(*
Nazwa:			P01_PucksInserter
Opis:			Stacja podajnika opakowań
Wersja:			v0.1
Data:			2025-02-04
Autor:			DP
Urzadzenia:		
Konfiguracja:	
Info:

*)
PROGRAM P01_PucksInserter
VAR_INPUT

	//52N6.1 Pneumatyka IO
	IbPucksInserterLevelSensor					:BOOL;			// Czujnik kolejki butelki
	IbPucksInserterWheelEntrySensor				:BOOL;			// Czujnik   pierwszego slotu w karuzeli (to 
	IbPucksInserterWheelExitSensor				:BOOL;			// Czujnik
	IbPucksInserterFormGateBeforeSensor 		:BOOL;			// Czujnik przed szlabanem formatek
	IbPucksInserterFormGateAfterSensor 			:BOOL;			// Czujnik za szlabanem formatek	
 	IbPucksInserterHammerUpSensor				:BOOL;			// Czujnik położenia siłownika - góra
	IbPucksInserterHammerDownSensor				:BOOL;			// Czujnik polożenia siłowniak - dół
	IbPucksInserterTrayOnSensor					:BOOL;			// Czujnik tacka wysunieta
	//52N6.2 Pneumatyka IO	
	IbPucksInserterTrayOffSensor				:BOOL;			// Czujnik tacka schowana
	IbPucksInserterFormPositioningOnSensor		:BOOL;			// Czujnik wysuniecia siłownika pozycjonujacego formatke
	IbPucksInserterFormPositioningOffSensor		:BOOL;			// Czujnik schowania siłownika pozycjonujacego formatke
	IbPucksInserterGate1OnSensor				:BOOL;			// Czujnik otwarcia 1 szlabanu (Lewy)
	IbPucksInserterGate1OffSensor				:BOOL;			// Czujnik zamknięcia 1 szlabanu (Lewy) 
	IbPucksInserterGate2OnSensor				:BOOL;			// Czujnik otwarcia 2 szlabanu 
	IbPucksInserterGate2OffSensor				:BOOL;			// Czujnik zamknięcia 2 szlabanu (Prawy) 
	IbPucksInserterHomingSensor					:BOOL;			// Czujnik bazowania
	
	//Inne
	IbPucksInserterNotInsertedSensor			:BOOL;			// Czujnik źle włozonej butelki za stacją	
	
	IbPucksInserterPushTablesSensor				:BOOL;
END_VAR

VAR

	//BC3 
	IbPucksInserterFuseDrivesOK					AT %I*: BOOL; 			// Zabezpieczenie serwa
	IbPucksInserterTransporter1OK				AT %I*: BOOL; 			// Bezpiecznik silnikowe napędu transportera 1
	IbPucksInserterTransporter2OK				AT %I*: BOOL; 			// Bezpiecznik silnikowe napędu transportera 2	
	IbPucksInserterFuseFB1OK					AT %I*: BOOL;			// Bezpiecznik FB1 przepalony
	QbPucksInserterHammerHeightUpCmd 			AT %Q*: BOOL; 			// Wyjście sterujące podnośnikiem
	QbPucksInserterHammerHeightDownCmd 			AT %Q*: BOOL; 			// Wyjście sterujące podnośnikiem
	//GVL_IO QbPickInserterDoorsClose			AT %Q*:BOOL;			// Rozkaz zamkniecia
	QudiPucksInserterHammerHeightEncoderSetCV	AT %Q*: UDINT;			// Enkoder - Set Counter value
	QbPucksInserterHammerHeightEncoderSetC		AT %Q*: BOOL; 			// Enkoder - Set Counter 
	IudiPucksInserterHammerHeightEncoderCV 		AT %I*: UDINT;	 		// Enkoder - Counter value
	IbPucksInserterHammerHeightEncoderSetCDone	AT %I*: BOOL; 			// Enkoder - Set Counter done

	//DI5
	//GVL_IO IbPucksInserterDoorsOpen	{warning 'PI'}	AT %I*	:BOOL;	//Otwarte drzwi podajnika opakowań
	//GLV_IO etop 0
	//GLV_IO etop 1
	//GLV_IO stop
	//GLV_IO start
	//Safety reset

	//DO4
	//Lamps green
	//Lamps blue

	fbPucksInserter						  	: FB_PucksInserter;		// Bloczek do obsługi stacji podajnika butelek
	fbTurnTable								: FB_MitsubishiInverter; 	//Bloczek do obsługi falownika stołu obrotewego
	
	ePucksInserterStationState				: E_Station;
	ePucksInserterRunningState				: E_PuckInserterState;
	fbPucksInserterState					: FB_State;
	
	ePucksInserterTurnTableState			: E_Station;
	ePucksInserterTurnTableRunningState		: E_ConveyorState;
	fbBottleSorterTurnTableState			: FB_State;
	
	fbGatePucksInserter						: FB_SpringGateV2;
	
	//Wyjścia sterujące
	QbPucksInserterHammer					:BOOL;			// Wbijak
	QbPucksInserterTray						:BOOL;			// Ruchomy blat (tacka)
	QbPucksInserterGate1					:BOOL;			// Szlaban 1 (lewy)
	QbPucksInserterGate2					:BOOL;			// Szlaban 2 (prawy)
	QbPucksInserterFormGate					:BOOL;			// Szlaban formatki
	QbPucksInserterFormPositioning			:BOOL;			// Pozycjonowanie formatki

	// Stół obrotowy
	uiPucksInserterTurnTableSW					AT %I*: UINT;
	uiPucksInserterTurnTableActualVelocity		AT %I*: UDINT;
	uiPucksInserterTurnTableCW  				AT %Q*: UINT;
	udiPucksInserterTurnTableVelocity			AT %Q*: UDINT;
	
	// Transporter
	uiPucksInserterConveyorSW					AT %I*: UINT;
	uiPucksInserterConveyorActualVelocity		AT %I*: UDINT;
	uiPucksInserterConveyorCW  					AT %Q*: UINT;
	udiPucksInserterConveyorVelocity			AT %Q*: UDINT;	
	IbPucksInserterConveyorWcState				AT %I*: BOOL;
	
	// Serwo
	// GVL axis
	diPucksInserterWheelZPhaseOffset			AT %I*: DINT; // Offset serwa Z


	// Bazowanie
	tonPucksInserterEnable	: TON;
	rtEnable	: R_TRIG;
	
	//testowe
	bTest :BOOL;
	bTest2 :BOOL;	
	bTestHomingPI:BOOL;
	bPITest:BOOL;
	 
	//Stół pchający    //Vasyl 27.05
	fbPushTable_m1: FB_MitsubishiInverter;
	fbPushTable_m2: FB_MitsubishiInverter;
	fbPushTable_m3: FB_MitsubishiInverter;	
	
	QnPucksInserterPushTable_m1_VelocitySV 						AT %Q*: UDINT; 	
	InPucksInserterPushTable_m1_VelocityCV 						AT %I*: UDINT;	
	InPucksInserterPushTable_m1_STW 							AT %I*: UINT; 	
	QnPucksInserterPushTable_m1_CTW 							AT %Q*: UINT;  	
	InPucksInserterPushTable_m1_ErrorCode 						AT %I*: UINT;	
	
	QnPucksInserterPushTable_m2_VelocitySV 						AT %Q*: UDINT; 	
	InPucksInserterPushTable_m2_VelocityCV 						AT %I*: UDINT;	
	InPucksInserterPushTable_m2_STW 							AT %I*: UINT; 
	QnPucksInserterPushTable_m2_CTW 							AT %Q*: UINT;  	
	InPucksInserterPushTable_m2_ErrorCode 						AT %I*: UINT;	
	
	QnPucksInserterPushTable_m3_VelocitySV 						AT %Q*: UDINT; 	
	InPucksInserterPushTable_m3_VelocityCV 						AT %I*: UDINT; 	
	InPucksInserterPushTable_m3_STW 							AT %I*: UINT; 
	QnPucksInserterPushTable_m3_CTW 							AT %Q*: UINT;  	
	InPucksInserterPushTable_m3_ErrorCode 						AT %I*: UINT;	

	
	fbPucksInserterPushTableState			: FB_State;
	ePucksInserterPushTableState			: E_Station;
	ePucksInserterPushTableRunningState		: E_PuckInserterState;
	
	fbPucksInserterPushTableRollerState			: FB_State;
	ePucksInserterPushTableRollerState			: E_Station;
	ePucksInserterPushTableRollerRunningState	: E_PuckInserterState;
END_VAR

aWarning();
aPucksInserter();
aTurntable(); 
aGateTime();
aGate();
aPushTable();

//VIS.nPucksInserterTurnTableVelocityCV := uiPucksInserterTurnTableActualVelocity;
VIS.nPucksInserterConveyorVelocityCV:=uiPucksInserterConveyorActualVelocity;
VIS.uiPucksInserterPushTable_m1_Velocity:=UDINT_TO_INT(InPucksInserterPushTable_m1_VelocityCV);
VIS.uiPucksInserterPushTable_m2_Velocity:=UDINT_TO_INT(InPucksInserterPushTable_m2_VelocityCV);
VIS.uiPucksInserterPushTable_m3_Velocity:=UDINT_TO_INT(InPucksInserterPushTable_m3_VelocityCV);

(* BAZOWANIE - ZMIAN*)
tonPucksInserterEnable (IN:=fbPucksInserter.bEnable,PT:=T#5S); (*Dodany ton bo Wizka zjebnie wgrywa zmienne, najpierw włacza Enabla a potem dopiero wybiera recepture*)
rtEnable(CLK:=tonPucksInserterEnable.Q,Q=>);
IF rtEnable.Q AND (P00_PackML.fbPMLAuto.ePMLState = E_PMLState.ePMLState_IDLE OR P00_PackML.fbPMLAuto.ePMLState = E_PMLState.ePMLState_EXECUTE)   THEN
	VIS.bPucksInserterHeightSet:=TRUE;
ELSIF fbPucksInserter.eState=E_Station.eHomingDone  OR VIS.bErrorOccure THEN
 	VIS.bPucksInserterHeightSet:=FALSE;
END_IF
(*KONIEC BAZOWANIE - ZMIANA*)


(********KASOWANIE ROZKAZÓW CYKLI*********)
IF fbPucksInserter.bCycleDone AND bManualMode THEN
	VIS.bPucksInserterRun := FALSE;
END_IF

(*
IF bPITest AND NOT VIS.bPucksInserterRun THEN
	VIS.bPucksInserterRun := TRUE;
END_IF
IF VIS.bPucksInserterRun AND bPITest AND fbPucksInserter.bCycleDone THEN
	VIS.bPucksInserterRun := FALSE;	
END_IF*)


fbPucksInserterState(
	eState									:= ePucksInserterStationState,
	bRun									:= VIS.bPucksInserterRun,
	eBottleSorterRunningState				:= ePucksInserterRunningState,
	sStateDesc								=> VIS.sPucksInserterState,
	iState									=> VIS.iPucksInserterState);
	
fbPucksInserterPushtableState(
	eState									:= ePucksInserterPushTableState,
    bRun						            := gvl.bPucksInserterPushTable_m1_Run OR vis.bPucksInserterPushTable_m1_ManualCmdStart,
    eBottleSorterRunningState	            := ePucksInserterPushTableRunningState,
    sStateDesc					            => VIS.sPucksInserterPushTableState,
    iState						            => VIS.iPucksInserterPushTableState);
	
fbPucksInserterPushTableRollerState(
	eState									:= ePucksInserterPushTableRollerState,	
    bRun						            := gvl.bPucksInserterPushTable_m2_Run OR vis.bPucksInserterPushTable_m2_ManualCmdStart,	
    eBottleSorterRunningState	            := ePucksInserterPushTableRollerRunningState,	
    sStateDesc					            => VIS.sPucksInserterPushTableRollerState,	
    iState						            => VIS.iPucksInserterPushTableRollerState);

ACTION aGate:
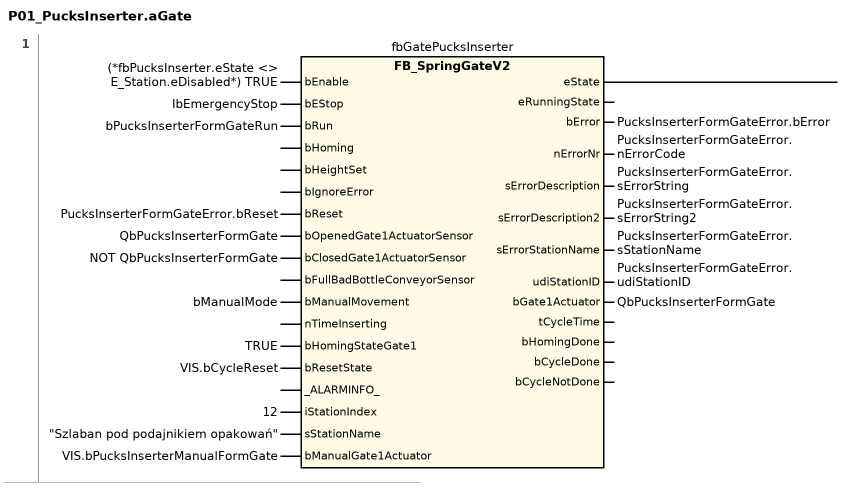
// NETWORK 1
fbGatePucksInserter(
    bEnable := (*fbPucksInserter.eState <> E_Station.eDisabled*) TRUE,
    bEStop := IbEmergencyStop,
    bRun := bPucksInserterFormGateRun,
    bReset := PucksInserterFormGateError.bReset,
    bOpenedGate1ActuatorSensor := QbPucksInserterFormGate,
    bClosedGate1ActuatorSensor := NOT QbPucksInserterFormGate,
    bManualMovement := bManualMode,
    bHomingStateGate1 := TRUE,
    bResetState := VIS.bCycleReset,
    iStationIndex := 12,
    sStationName := "Szlaban pod podajnikiem opakowań",
    bManualGate1Actuator := VIS.bPucksInserterManualFormGate,
    bError => PucksInserterFormGateError.bError,
    nErrorNr => PucksInserterFormGateError.nErrorCode,
    sErrorDescription => PucksInserterFormGateError.sErrorString,
    sErrorDescription2 => PucksInserterFormGateError.sErrorString2,
    sErrorStationName => PucksInserterFormGateError.sStationName,
    udiStationID => PucksInserterFormGateError.udiStationID,
    bGate1Actuator => QbPucksInserterFormGate); // FB_SpringGateV2
END_ACTION

ACTION aGateTime:
IF bFormTransportersDispencerSlowSpeed THEN 
	fbGatePucksInserter.nTimeInserting	:=	350; //500 pomieszane zwalnianie transportera??
ELSE
	fbGatePucksInserter.nTimeInserting	:=	350;	//400
END_IF
END_ACTION

ACTION aPucksInserter:
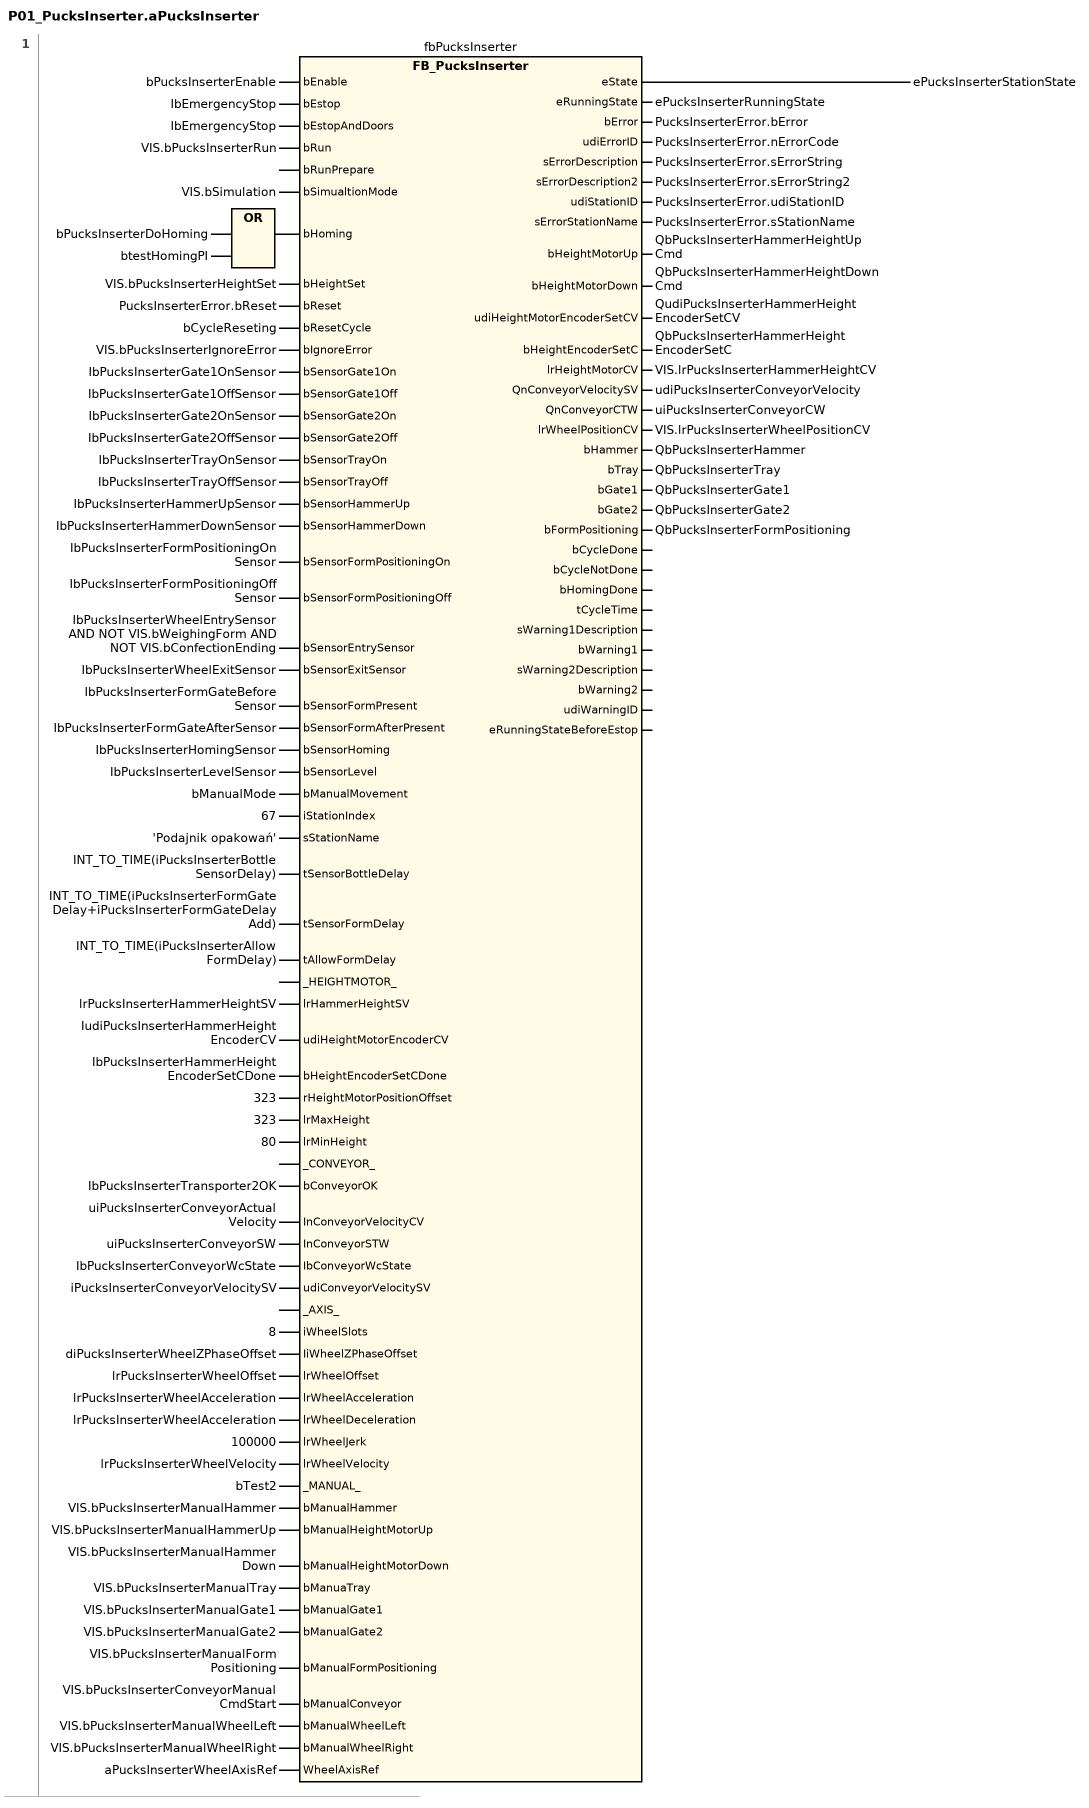
// NETWORK 1
fbPucksInserter(
    bEnable := bPucksInserterEnable,
    bEstop := IbEmergencyStop,
    bEstopAndDoors := IbEmergencyStop,
    bRun := VIS.bPucksInserterRun,
    bSimualtionMode := VIS.bSimulation,
    bHoming := bPucksInserterDoHoming OR btestHomingPI,
    bHeightSet := VIS.bPucksInserterHeightSet,
    bReset := PucksInserterError.bReset,
    bResetCycle := bCycleReseting,
    bIgnoreError := VIS.bPucksInserterIgnoreError,
    bSensorGate1On := IbPucksInserterGate1OnSensor,
    bSensorGate1Off := IbPucksInserterGate1OffSensor,
    bSensorGate2On := IbPucksInserterGate2OnSensor,
    bSensorGate2Off := IbPucksInserterGate2OffSensor,
    bSensorTrayOn := IbPucksInserterTrayOnSensor,
    bSensorTrayOff := IbPucksInserterTrayOffSensor,
    bSensorHammerUp := IbPucksInserterHammerUpSensor,
    bSensorHammerDown := IbPucksInserterHammerDownSensor,
    bSensorFormPositioningOn := IbPucksInserterFormPositioningOnSensor,
    bSensorFormPositioningOff := IbPucksInserterFormPositioningOffSensor,
    bSensorEntrySensor := IbPucksInserterWheelEntrySensor AND NOT VIS.bWeighingForm AND NOT VIS.bConfectionEnding,
    bSensorExitSensor := IbPucksInserterWheelExitSensor,
    bSensorFormPresent := IbPucksInserterFormGateBeforeSensor,
    bSensorFormAfterPresent := IbPucksInserterFormGateAfterSensor,
    bSensorHoming := IbPucksInserterHomingSensor,
    bSensorLevel := IbPucksInserterLevelSensor,
    bManualMovement := bManualMode,
    iStationIndex := 67,
    sStationName := 'Podajnik opakowań',
    tSensorBottleDelay := INT_TO_TIME(iPucksInserterBottleSensorDelay),
    tSensorFormDelay := INT_TO_TIME(iPucksInserterFormGateDelay+iPucksInserterFormGateDelayAdd),
    tAllowFormDelay := INT_TO_TIME(iPucksInserterAllowFormDelay),
    lrHammerHeightSV := lrPucksInserterHammerHeightSV,
    udiHeightMotorEncoderCV := IudiPucksInserterHammerHeightEncoderCV,
    bHeightEncoderSetCDone := IbPucksInserterHammerHeightEncoderSetCDone,
    rHeightMotorPositionOffset := 323,
    lrMaxHeight := 323,
    lrMinHeight := 80,
    bConveyorOK := IbPucksInserterTransporter2OK,
    InConveyorVelocityCV := uiPucksInserterConveyorActualVelocity,
    InConveyorSTW := uiPucksInserterConveyorSW,
    IbConveyorWcState := IbPucksInserterConveyorWcState,
    udiConveyorVelocitySV := iPucksInserterConveyorVelocitySV,
    iWheelSlots := 8,
    IiWheelZPhaseOffset := diPucksInserterWheelZPhaseOffset,
    lrWheelOffset := lrPucksInserterWheelOffset,
    lrWheelAcceleration := lrPucksInserterWheelAcceleration,
    lrWheelDeceleration := lrPucksInserterWheelAcceleration,
    lrWheelJerk := 100000,
    lrWheelVelocity := lrPucksInserterWheelVelocity,
    _MANUAL_ := bTest2,
    bManualHammer := VIS.bPucksInserterManualHammer,
    bManualHeightMotorUp := VIS.bPucksInserterManualHammerUp,
    bManualHeightMotorDown := VIS.bPucksInserterManualHammerDown,
    bManuaTray := VIS.bPucksInserterManualTray,
    bManualGate1 := VIS.bPucksInserterManualGate1,
    bManualGate2 := VIS.bPucksInserterManualGate2,
    bManualFormPositioning := VIS.bPucksInserterManualFormPositioning,
    bManualConveyor := VIS.bPucksInserterConveyorManualCmdStart,
    bManualWheelLeft := VIS.bPucksInserterManualWheelLeft,
    bManualWheelRight := VIS.bPucksInserterManualWheelRight,
    WheelAxisRef := aPucksInserterWheelAxisRef,
    eRunningState => ePucksInserterRunningState,
    bError => PucksInserterError.bError,
    udiErrorID => PucksInserterError.nErrorCode,
    sErrorDescription => PucksInserterError.sErrorString,
    sErrorDescription2 => PucksInserterError.sErrorString2,
    udiStationID => PucksInserterError.udiStationID,
    sErrorStationName => PucksInserterError.sStationName,
    bHeightMotorUp => QbPucksInserterHammerHeightUpCmd,
    bHeightMotorDown => QbPucksInserterHammerHeightDownCmd,
    udiHeightMotorEncoderSetCV => QudiPucksInserterHammerHeightEncoderSetCV,
    bHeightEncoderSetC => QbPucksInserterHammerHeightEncoderSetC,
    lrHeightMotorCV => VIS.lrPucksInserterHammerHeightCV,
    QnConveyorVelocitySV => udiPucksInserterConveyorVelocity,
    QnConveyorCTW => uiPucksInserterConveyorCW,
    lrWheelPositionCV => VIS.lrPucksInserterWheelPositionCV,
    bHammer => QbPucksInserterHammer,
    bTray => QbPucksInserterTray,
    bGate1 => QbPucksInserterGate1,
    bGate2 => QbPucksInserterGate2,
    bFormPositioning => QbPucksInserterFormPositioning); // FB_PucksInserter
ePucksInserterStationState := fbPucksInserter.eState;
END_ACTION

ACTION aPushTable:
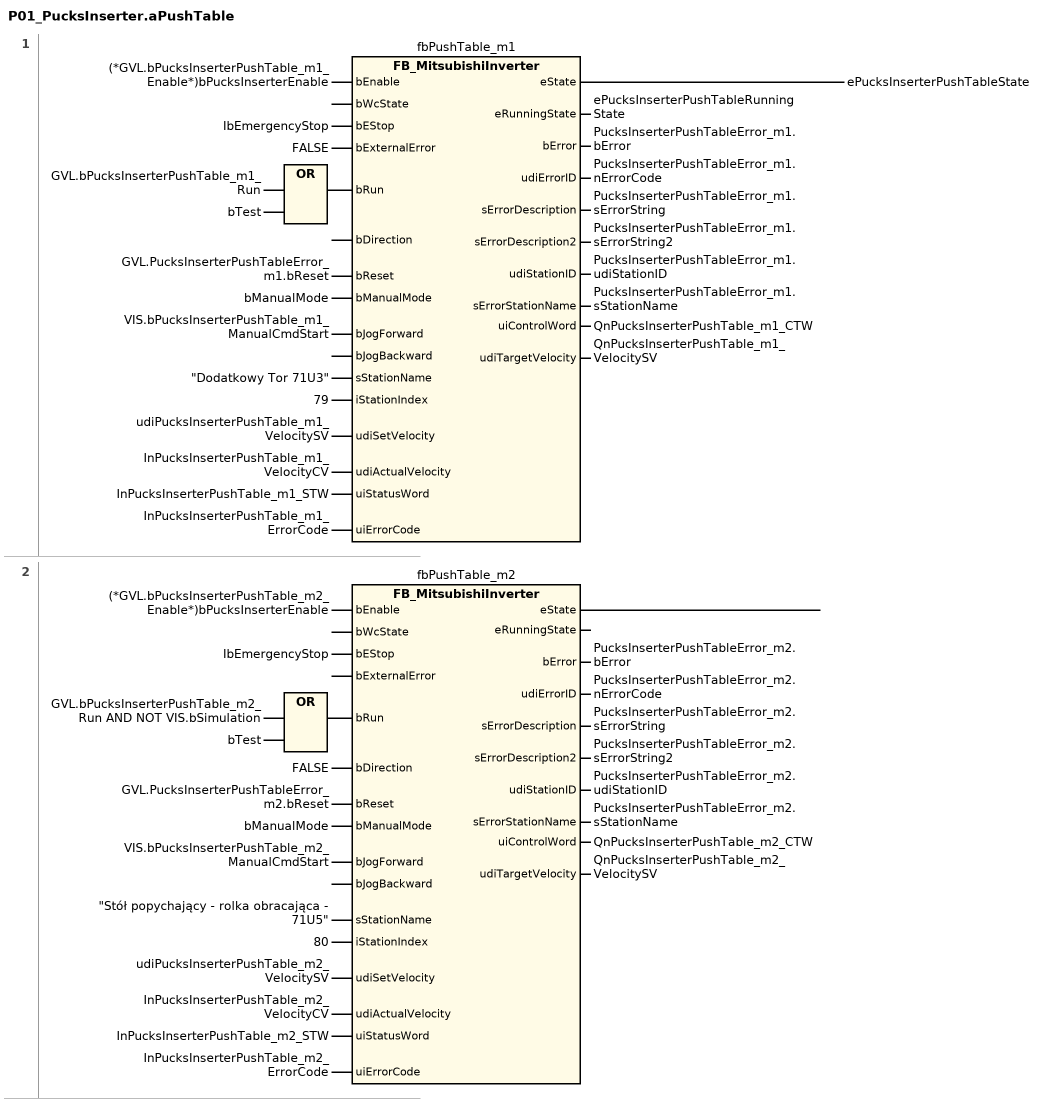
// NETWORK 1
fbPushTable_m1(
    bEnable := (*GVL.bPucksInserterPushTable_m1_Enable*)bPucksInserterEnable,
    bEStop := IbEmergencyStop,
    bExternalError := FALSE,
    bRun := GVL.bPucksInserterPushTable_m1_Run OR bTest,
    bReset := GVL.PucksInserterPushTableError_m1.bReset,
    bManualMode := bManualMode,
    bJogForward := VIS.bPucksInserterPushTable_m1_ManualCmdStart,
    sStationName := "Dodatkowy Tor 71U3",
    iStationIndex := 79,
    udiSetVelocity := udiPucksInserterPushTable_m1_VelocitySV,
    udiActualVelocity := InPucksInserterPushTable_m1_VelocityCV,
    uiStatusWord := InPucksInserterPushTable_m1_STW,
    uiErrorCode := InPucksInserterPushTable_m1_ErrorCode,
    eRunningState => ePucksInserterPushTableRunningState,
    bError => PucksInserterPushTableError_m1.bError,
    udiErrorID => PucksInserterPushTableError_m1.nErrorCode,
    sErrorDescription => PucksInserterPushTableError_m1.sErrorString,
    sErrorDescription2 => PucksInserterPushTableError_m1.sErrorString2,
    udiStationID => PucksInserterPushTableError_m1.udiStationID,
    sErrorStationName => PucksInserterPushTableError_m1.sStationName,
    uiControlWord => QnPucksInserterPushTable_m1_CTW,
    udiTargetVelocity => QnPucksInserterPushTable_m1_VelocitySV); // FB_MitsubishiInverter
ePucksInserterPushTableState := fbPushTable_m1.eState;

// NETWORK 2
fbPushTable_m2(
    bEnable := (*GVL.bPucksInserterPushTable_m2_Enable*)bPucksInserterEnable,
    bEStop := IbEmergencyStop,
    bRun := (GVL.bPucksInserterPushTable_m2_Run AND NOT VIS.bSimulation) OR bTest,
    bDirection := FALSE,
    bReset := GVL.PucksInserterPushTableError_m2.bReset,
    bManualMode := bManualMode,
    bJogForward := VIS.bPucksInserterPushTable_m2_ManualCmdStart,
    sStationName := "Stół popychający - rolka obracająca - 71U5",
    iStationIndex := 80,
    udiSetVelocity := udiPucksInserterPushTable_m2_VelocitySV,
    udiActualVelocity := InPucksInserterPushTable_m2_VelocityCV,
    uiStatusWord := InPucksInserterPushTable_m2_STW,
    uiErrorCode := InPucksInserterPushTable_m2_ErrorCode,
    bError => PucksInserterPushTableError_m2.bError,
    udiErrorID => PucksInserterPushTableError_m2.nErrorCode,
    sErrorDescription => PucksInserterPushTableError_m2.sErrorString,
    sErrorDescription2 => PucksInserterPushTableError_m2.sErrorString2,
    udiStationID => PucksInserterPushTableError_m2.udiStationID,
    sErrorStationName => PucksInserterPushTableError_m2.sStationName,
    uiControlWord => QnPucksInserterPushTable_m2_CTW,
    udiTargetVelocity => QnPucksInserterPushTable_m2_VelocitySV); // FB_MitsubishiInverter

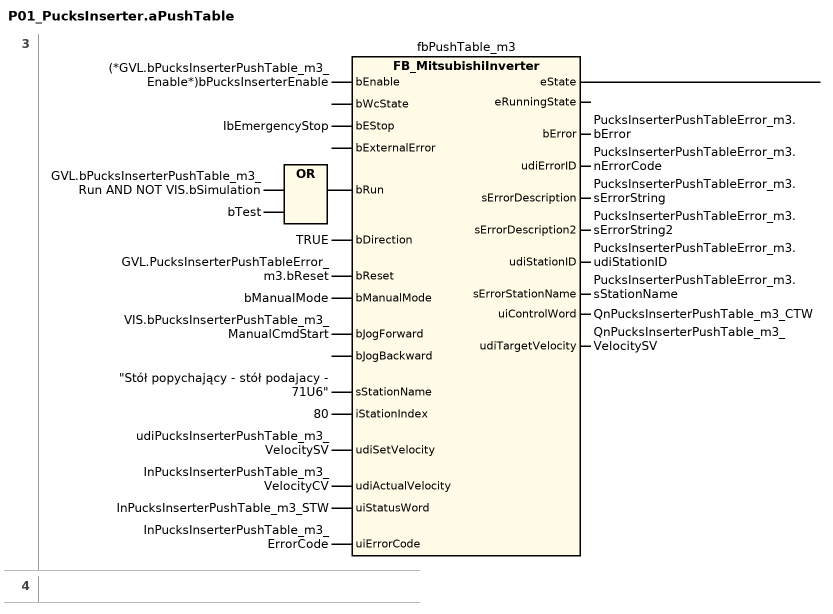
// NETWORK 3
fbPushTable_m3(
    bEnable := (*GVL.bPucksInserterPushTable_m3_Enable*)bPucksInserterEnable,
    bEStop := IbEmergencyStop,
    bRun := (GVL.bPucksInserterPushTable_m3_Run AND NOT VIS.bSimulation) OR bTest,
    bDirection := TRUE,
    bReset := GVL.PucksInserterPushTableError_m3.bReset,
    bManualMode := bManualMode,
    bJogForward := VIS.bPucksInserterPushTable_m3_ManualCmdStart,
    sStationName := "Stół popychający - stół podajacy - 71U6",
    iStationIndex := 80,
    udiSetVelocity := udiPucksInserterPushTable_m3_VelocitySV,
    udiActualVelocity := InPucksInserterPushTable_m3_VelocityCV,
    uiStatusWord := InPucksInserterPushTable_m3_STW,
    uiErrorCode := InPucksInserterPushTable_m3_ErrorCode,
    bError => PucksInserterPushTableError_m3.bError,
    udiErrorID => PucksInserterPushTableError_m3.nErrorCode,
    sErrorDescription => PucksInserterPushTableError_m3.sErrorString,
    sErrorDescription2 => PucksInserterPushTableError_m3.sErrorString2,
    udiStationID => PucksInserterPushTableError_m3.udiStationID,
    sErrorStationName => PucksInserterPushTableError_m3.sStationName,
    uiControlWord => QnPucksInserterPushTable_m3_CTW,
    udiTargetVelocity => QnPucksInserterPushTable_m3_VelocitySV); // FB_MitsubishiInverter

// NETWORK 4
END_ACTION

ACTION aTurntable:
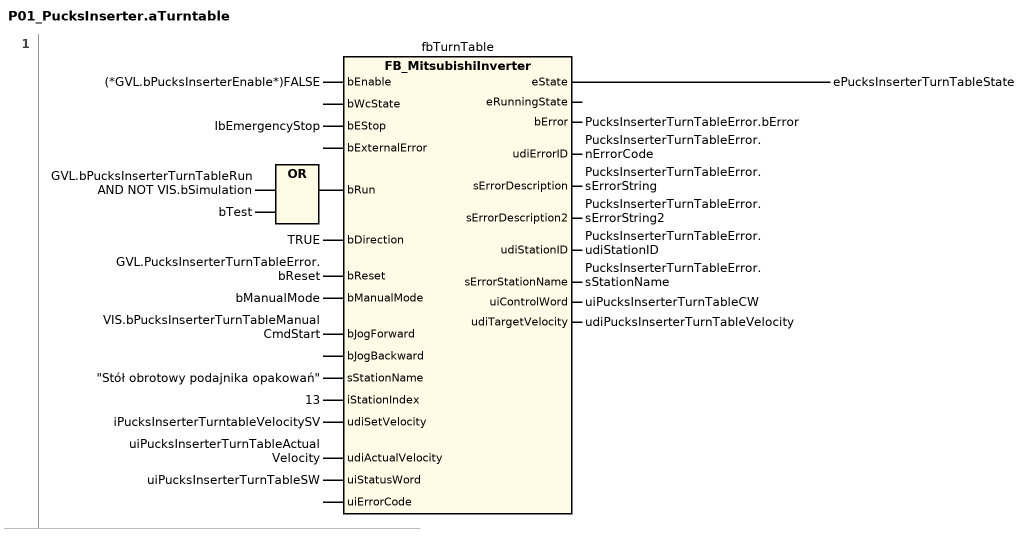
// NETWORK 1
fbTurnTable(
    bEnable := (*GVL.bPucksInserterEnable*)FALSE,
    bEStop := IbEmergencyStop,
    bRun := (GVL.bPucksInserterTurnTableRun AND NOT VIS.bSimulation) OR bTest,
    bDirection := TRUE,
    bReset := GVL.PucksInserterTurnTableError.bReset,
    bManualMode := bManualMode,
    bJogForward := VIS.bPucksInserterTurnTableManualCmdStart,
    sStationName := "Stół obrotowy podajnika opakowań",
    iStationIndex := 13,
    udiSetVelocity := iPucksInserterTurntableVelocitySV,
    udiActualVelocity := uiPucksInserterTurnTableActualVelocity,
    uiStatusWord := uiPucksInserterTurnTableSW,
    bError => PucksInserterTurnTableError.bError,
    udiErrorID => PucksInserterTurnTableError.nErrorCode,
    sErrorDescription => PucksInserterTurnTableError.sErrorString,
    sErrorDescription2 => PucksInserterTurnTableError.sErrorString2,
    udiStationID => PucksInserterTurnTableError.udiStationID,
    sErrorStationName => PucksInserterTurnTableError.sStationName,
    uiControlWord => uiPucksInserterTurnTableCW,
    udiTargetVelocity => udiPucksInserterTurnTableVelocity); // FB_MitsubishiInverter
ePucksInserterTurnTableState := fbTurnTable.eState;
END_ACTION

ACTION aWarning:
// Warning 1
IF (IbBottleFeederSafetyDoor3Open AND bPucksInserterEnable) AND NOT BottleFeederWarning[0].bWarning THEN
	BottleFeederWarning[0].bWarning										:=TRUE;
	BottleFeederWarning[0].udiWarningCode								:=1;
	BottleFeederWarning[0].sDescription									:='Podajnik butelek | Otwarte drzwi dostępowe';
ELSIF (NOT GVL_io.IbBottleFeederSafetyDoor3Open OR NOT bPucksInserterEnable) (*AND PucksInserterWarning[0].bAcknowledge*) THEN
	BottleFeederWarning[0].bWarning										:= FALSE;
	BottleFeederWarning[0].bAcknowledge									:= FALSE;
	VIS.uliWarningAcknowledge.23 										:= FALSE;
//ELSIF PucksInserterWarning[0].bAcknowledge THEN
//ELSE
//	PucksInserterWarning[0].bAcknowledge									:= TRUE;
END_IF	

// Warning 2

IF (fbPucksInserter.bWarning1 AND bPucksInserterEnable) AND NOT BottleFeederWarning[1].bWarning THEN
	BottleFeederWarning[1].bWarning										:= TRUE;
	BottleFeederWarning[1].udiWarningCode								:= 2;
	BottleFeederWarning[1].sDescription									:= 'Podajnik butelek | Niski poziom butelek';
ELSIF (NOT fbPucksInserter.bWarning1 OR NOT bPucksInserterEnable) (*AND BottleFeederWarning[1].bAcknowledge*) THEN
	BottleFeederWarning[1].bWarning										:= FALSE;
	BottleFeederWarning[1].bAcknowledge									:= FALSE;
	VIS.uliWarningAcknowledge.26 										:= FALSE;
ELSIF BottleFeederWarning[1].bAcknowledge THEN
	BottleFeederWarning[1].bAcknowledge									:= TRUE;
END_IF

//Warning 3
IF (IbBottleFeederSafetyDoor1Open AND bPucksInserterEnable) AND NOT BottleFeederWarning[2].bWarning THEN
	BottleFeederWarning[2].bWarning										:=TRUE;
	BottleFeederWarning[2].udiWarningCode								:=3;
	BottleFeederWarning[2].sDescription									:='Podajnik butelek | Otwarta bramka wjazdowa';
ELSIF (NOT IbBottleFeederSafetyDoor1Open OR NOT bPucksInserterEnable) (*AND BottleFeederWarning[2].bAcknowledge*) THEN
	BottleFeederWarning[2].bWarning										:= FALSE;
	BottleFeederWarning[2].bAcknowledge									:= FALSE;
	VIS.uliWarningAcknowledge.41 										:= FALSE;
//ELSIF BottleFeederWarning[2].bAcknowledge THEN
//	BottleFeederWarning[2].bAcknowledge									:= TRUE;
END_IF	

//Warning 4
BottleFeederWarning[3].sDescription										:='Podajnik butelek | Otwarta bramka wyjazdowa';
IF (IbBottleFeederSafetyDoor2Open AND bPucksInserterEnable) AND NOT BottleFeederWarning[3].bWarning THEN
	BottleFeederWarning[3].bWarning										:=TRUE;
	BottleFeederWarning[3].udiWarningCode								:=4;
	BottleFeederWarning[3].sDescription									:='Podajnik butelek | Otwarta bramka wyjazdowa';
ELSIF (NOT GVL_io.IbBottleFeederSafetyDoor2Open OR NOT bPucksInserterEnable) (*AND BottleFeederWarning[3].bAcknowledge*) THEN
	BottleFeederWarning[3].bWarning										:= FALSE;
	BottleFeederWarning[3].bAcknowledge									:= FALSE;
	VIS.uliWarningAcknowledge.42 										:= FALSE;
//ELSIF BottleFeederWarning[3].bAcknowledge THEN
//	BottleFeederWarning[3].bAcknowledge									:= TRUE;
END_IF
END_ACTION

END_PROGRAM

(* stored: Version 1.2.0.0, ProductVersion 3.1.4026.13, FileIdentifier b5083c7843d65664c7e280660fdfab420d28fa35, FileSignature 65850fdd5d6f50819ecb4cab93d0035f8d8a46bab9924d1756ebb6b863742ac0ffa6bddab7329a2441d152f2e46cb82ba21c51b1c79c19d2aedcd1996ef19080f1f9ecd2054d695b78a0e867380740fedb5d575761fe5df5e1fd5c3e919c06611cee44fe5c91bdcdc19f671871284a9045bb44682fea1388be577ca65cfe8cebc1dd59d5bd13737f12fe07e5d1e81d3325a734b7aaf29cb759eee9c2c50fbdd10755019062cbe6cab164b450dec77457fa05e00521d0b884d5fac44138ccaecaa90f3c042278d11b45e6d317861f13514f8896e88859b3c02eb73a95b77d065ec9c8e5b0ca62a10006a39c52092c2f8bc324c15e8ede77ccf088465a5aacafdd
   POU P01_PucksInserter: Id {8e20e43e-fe41-4397-9199-4cccbb867553}, SpecialFunc None
   Action aGate: Id {299f8aa8-3043-4c4f-b456-13a0eb95acd2}
   Action aGateTime: Id {2b8effef-4e6c-4b35-8dab-7c44ed28fa39}
   Action aPucksInserter: Id {dcaac96f-5870-4ebf-bad9-3d37583f1fa5}
   Action aPushTable: Id {9d87465f-49f6-4ff4-980e-c76a15a51f90}
   Action aTurntable: Id {cc87a089-bc86-4c28-8ea3-1fe0fcca284a}
   Action aWarning: Id {a5c23e82-5f3c-471e-90a0-8a80e09ececa} *)
